TYPE TupleStruct_3:
    STRUCT
        field0: BOOL;
        field1: BOOL;
        field2: BOOL;
        field3: BOOL;
        field4: BOOL;
        field5: BOOL;
        field6: BOOL;
        field7: BOOL;
        field8: BOOL;
        field9: BOOL;
        field10: BOOL;
        field11: BOOL;
        field12: BOOL;
        field13: BOOL;
        field14: BOOL;
        field15: BOOL;
        field16: BOOL;
        field17: BOOL;
        field18: BOOL;
        field19: BOOL;
        field20: BOOL;
        field21: BOOL;
        field22: BOOL;
        field23: BOOL;
        field24: BOOL;
        field25: BOOL;
        field26: BOOL;
        field27: BOOL;
        field28: BOOL;
        field29: BOOL;
        field30: BOOL;
        field31: BOOL;
        field32: BOOL;
        field33: BOOL;
        field34: BOOL;
        field35: BOOL;
        field36: BOOL;
        field37: BOOL;
        field38: BOOL;
        field39: BOOL;
        field40: BOOL;
        field41: BOOL;
        field42: BOOL;
        field43: BOOL;
        field44: BOOL;
        field45: BOOL;
        field46: BOOL;
        field47: BOOL;
        field48: BOOL;
        field49: BOOL;
        field50: BOOL;
        field51: BOOL;
        field52: BOOL;
        field53: BOOL;
        field54: BOOL;
        field55: BOOL;
        field56: BOOL;
        field57: BOOL;
        field58: BOOL;
        field59: BOOL;
        field60: BOOL;
        field61: BOOL;
        field62: BOOL;
        field63: BOOL;
        field64: BOOL;
        field65: BOOL;
        field66: BOOL;
        field67: BOOL;
        field68: BOOL;
        field69: BOOL;
        field70: BOOL;
        field71: BOOL;
        field72: BOOL;
        field73: BOOL;
        field74: BOOL;
        field75: BOOL;
        field76: BOOL;
        field77: BOOL;
        field78: BOOL;
        field79: BOOL;
        field80: BOOL;
        field81: BOOL;
        field82: BOOL;
        field83: BOOL;
        field84: BOOL;
        field85: BOOL;
        field86: BOOL;
        field87: BOOL;
        field88: BOOL;
        field89: BOOL;
        field90: BOOL;
        field91: BOOL;
        field92: BOOL;
        field93: BOOL;
        field94: BOOL;
        field95: BOOL;
        field96: BOOL;
        field97: BOOL;
        field98: BOOL;
        field99: BOOL;
    END_STRUCT
END_TYPE

(* stored: ProductVersion 3.1.0.18, Version 1.1.0.1 *)
